// TIA Portal V19 export
TYPE "PositioningMachine_Ax_Parameters"
// stored: Access Published
   STRUCT
      EncoderInverseDirection : Bool;
      MotorInverseDirection : Bool;
      LoadGearNumerator : UDInt;
      LoadGearDenominator : UDInt;
      MechanicsLeadScrew : LReal;
      EncoderDistancePerRevolution : LReal;
      DynamicsLimitsMaxVelocity : LReal;
      DynamicsLimitsVelocity : LReal;
      ControlLoop_Kv : LReal;
      ControlLoop_Kpc : LReal;
      ControlLoop_Vtc : LReal;
   END_STRUCT;
END_TYPE
